PROGRAM simulink_testing

VAR
	setTemp AT%Q*: LREAL;
	fdbkTemp AT%Q*: LREAL;
	power AT%I*: LREAL;
END_VAR

END_PROGRAM

(* stored: Version 1.1.0.1, ProductVersion 3.1.4024.13
   POU simulink_testing: Id {e8542fb9-a294-4c1b-89ab-317995b04a2f}, SpecialFunc None *)
